TYPE GearInPos_CMD_typ :
STRUCT
	StartSlave : BOOL ;
	DisengageSlave : BOOL ;
END_STRUCT
END_TYPE

(* stored: Version 1.1.0.1, ProductVersion 3.1.4024.3
   DUT GearInPos_CMD_typ: Id {abc87d9b-d3a3-0e0d-2d5a-036e3769d7b4} *)
